// Mitsubishi GX Works2 project: counter4   PLC: Q03UDV

PROGRAM MAIN
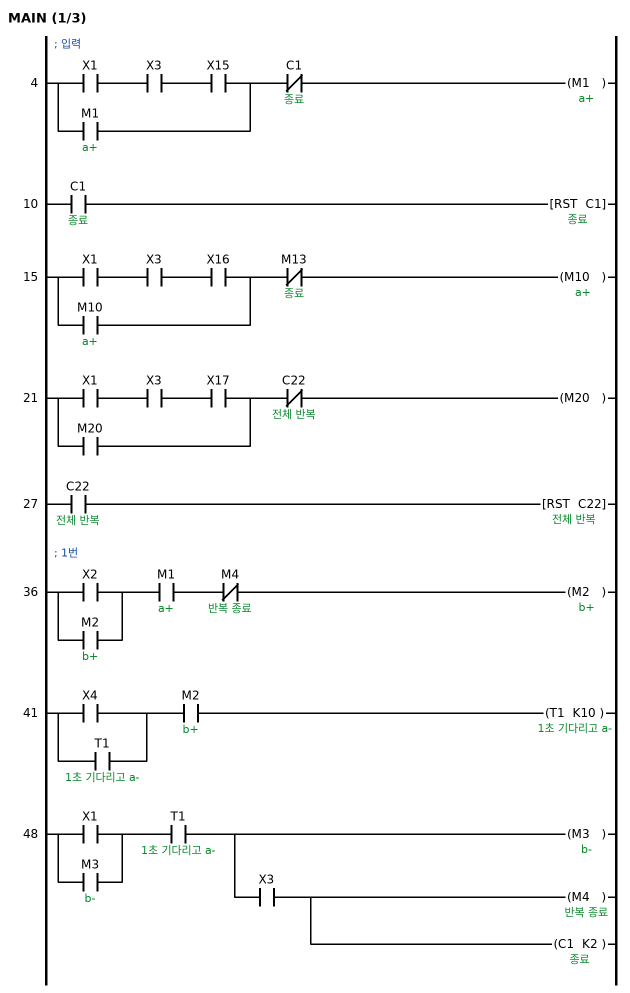
; 입력
4     LD      X1
      AND     X3
      AND     X15
      OR      M1  ; a+
      ANI     C1  ; 종료
      OUT     M1  ; a+
10    LD      C1  ; 종료
      RST     C1  ; 종료
15    LD      X1
      AND     X3
      AND     X16
      OR      M10  ; a+
      ANI     M13  ; 종료
      OUT     M10  ; a+
21    LD      X1
      AND     X3
      AND     X17
      OR      M20
      ANI     C22  ; 전체 반복
      OUT     M20
27    LD      C22  ; 전체 반복
      RST     C22  ; 전체 반복
; 1번
36    LD      X2
      OR      M2  ; b+
      AND     M1  ; a+
      ANI     M4  ; 반복 종료
      OUT     M2  ; b+
41    LD      X4
      OR      T1  ; 1초 기다리고 a-
      AND     M2  ; b+
      OUT     T1 K10  ; 1초 기다리고 a-
48    LD      X1
      OR      M3  ; b-
      AND     T1  ; 1초 기다리고 a-
      OUT     M3  ; b-
      AND     X3
      OUT     M4  ; 반복 종료
      OUT     C1 K2  ; 종료
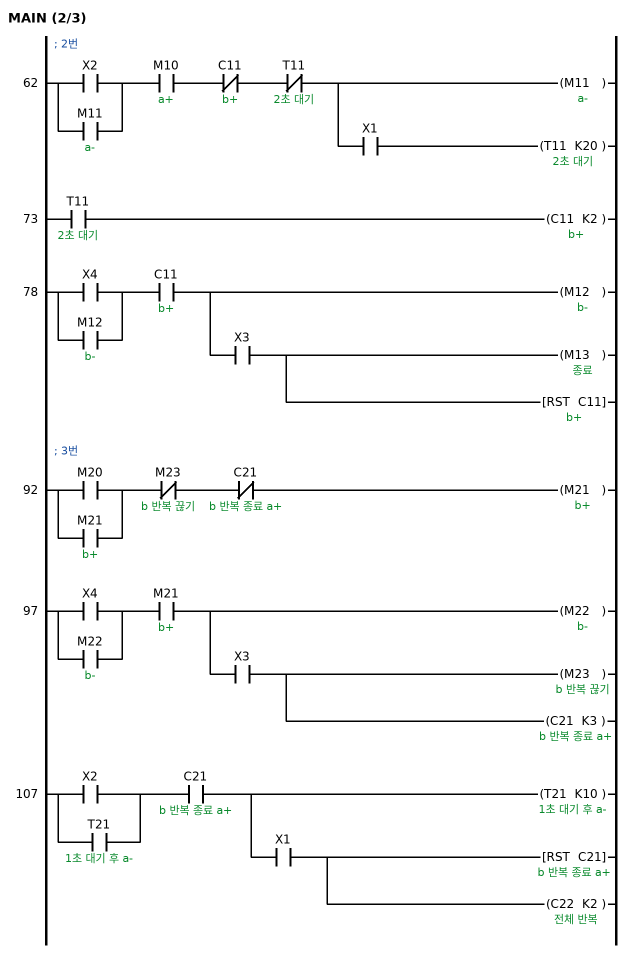
; 2번
62    LD      X2
      OR      M11  ; a-
      AND     M10  ; a+
      ANI     C11  ; b+
      ANI     T11  ; 2초 대기
      OUT     M11  ; a-
      AND     X1
      OUT     T11 K20  ; 2초 대기
73    LD      T11  ; 2초 대기
      OUT     C11 K2  ; b+
78    LD      X4
      OR      M12  ; b-
      AND     C11  ; b+
      OUT     M12  ; b-
      AND     X3
      OUT     M13  ; 종료
      RST     C11  ; b+
; 3번
92    LD      M20
      OR      M21  ; b+
      ANI     M23  ; b 반복 끊기
      ANI     C21  ; b 반복 종료 a+
      OUT     M21  ; b+
97    LD      X4
      OR      M22  ; b-
      AND     M21  ; b+
      OUT     M22  ; b-
      AND     X3
      OUT     M23  ; b 반복 끊기
      OUT     C21 K3  ; b 반복 종료 a+
107   LD      X2
      OR      T21  ; 1초 대기 후 a-
      AND     C21  ; b 반복 종료 a+
      OUT     T21 K10  ; 1초 대기 후 a-
      AND     X1
      RST     C21  ; b 반복 종료 a+
      OUT     C22 K2  ; 전체 반복
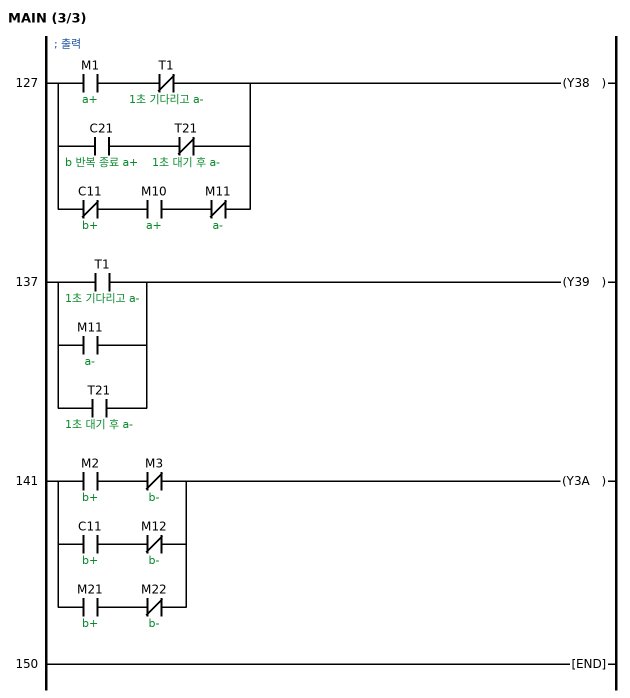
; 출력
127   LD      M1  ; a+
      ANI     T1  ; 1초 기다리고 a-
      LD      C21  ; b 반복 종료 a+
      ANI     T21  ; 1초 대기 후 a-
      ORB
      LDI     C11  ; b+
      AND     M10  ; a+
      ANI     M11  ; a-
      ORB
      OUT     Y38
137   LD      T1  ; 1초 기다리고 a-
      OR      M11  ; a-
      OR      T21  ; 1초 대기 후 a-
      OUT     Y39
141   LD      M2  ; b+
      ANI     M3  ; b-
      LD      C11  ; b+
      ANI     M12  ; b-
      ORB
      LD      M21  ; b+
      ANI     M22  ; b-
      ORB
      OUT     Y3A
150   END
END_PROGRAM

// device comments not shown above
M24  ; 전체 반복 끊기
